TYPE TxHmiLeica :
STRUCT
	status : DINT;
	x : REAL;
	y : REAL;
	z : REAL;
	q0 : REAL;
	q1 : REAL;
	q2 : REAL;
	q3 : REAL;
END_STRUCT
END_TYPE

(* stored: Version 1.1.0.1, ProductVersion 3.1.4020.12
   DUT TxHmiLeica: Id {3ac98ad6-ac07-43f2-b4f9-18ed0a1b7b2f} *)
